FUNCTION_BLOCK FB_VFD IMPLEMENTS I_Analog, I_Run
VAR_INPUT
END_VAR
VAR_OUTPUT
END_VAR
VAR
	_Coil 			: BOOL;
	_AnalogSignal 	: INT;
	_ScaledAnalog 	: INT;
END_VAR

{warning 'Agregar implementación de propiedad'}
PROPERTY AnalogSignal : INT
GET
AnalogSignal := _AnalogSignal;
END_GET
SET
_AnalogSignal := AnalogSignal;
END_SET
END_PROPERTY

{warning 'Agregar implementación de propiedad'}
PROPERTY Coil : BOOL
GET
Coil := _Coil;
END_GET
SET
_Coil := Coil;
END_SET
END_PROPERTY

{warning 'Agregar implementación de método'}
METHOD Scale : BOOL
ScaledAnalog := AnalogSignal * 200;
END_METHOD

{warning 'Agregar implementación de propiedad'}
PROPERTY ScaledAnalog : INT
GET
ScaledAnalog := _ScaledAnalog;
END_GET
SET
_ScaledAnalog := ScaledAnalog;
END_SET
END_PROPERTY

{warning 'Agregar implementación de método'}
METHOD Start : BOOL
Coil := true;
END_METHOD

{warning 'Agregar implementación de método'}
METHOD Stop : BOOL
Coil := false;
END_METHOD

END_FUNCTION_BLOCK

(* stored: Version 1.1.0.1, ProductVersion 3.1.4024.12
   POU FB_VFD: Id {ffc6ba41-6e19-4d67-9484-e64f63cbe576}, SpecialFunc None
   Property AnalogSignal: Id {31f78fa4-a832-42d2-ac65-0d96b1bba130}
   Get Get: Id {a632d7f8-e87e-437f-bf1d-6eae4906db64}
   Set Set: Id {9c840049-c3cb-42f5-af31-1824c15f449e}
   Property Coil: Id {fa8eb037-d6ab-4377-bff6-cc9476d5c0df}
   Get Get: Id {ca01a59b-b518-4a6d-bb2f-be6d82019541}
   Set Set: Id {386ffc64-7bb3-41b1-ad48-80e43c81d407}
   Method Scale: Id {01aea459-85a9-43f0-9c77-0790fff93e40}
   Property ScaledAnalog: Id {8d0b6189-b7fa-4f1d-a6a2-351ed9cdcc53}
   Get Get: Id {8eb1cc46-70ab-4c38-9988-795e01c9c5f3}
   Set Set: Id {4b66ed0f-a0d7-43f2-a1af-31bc04b99bbb}
   Method Start: Id {1a9ecbe1-0f1f-4a9b-b69e-97b9ca9075bb}
   Method Stop: Id {6f0e5fb1-6aa4-45be-ab90-5c7924fdb9e2} *)
